TYPE ST_LoggerSettings :
STRUCT
	netID : STRING(20);
	filePath : T_MaxString;
	filePrefix : STRING(10);
	FileType : STRING(10);
END_STRUCT
END_TYPE

(* stored: Version 1.1.0.1
   DUT ST_LoggerSettings: Id {cbd5a83d-7979-4719-b53b-191049e3be23} *)
